FUNCTION_BLOCK SchieberVerriegelung (* Schieber verriegeln bei 3 Schieber *)
  (* Standard: 61499-2; Description: Copyright (c) 2025 HR Agrartechnik GmbH This program and the accompanying materials are made available under the terms of the Eclipse Public License 2.0 which is available at https://www.eclipse.org/legal/epl-2.0/ SPDX-License-Identifier: EPL-2.0 *)
  (* Version 1.0, 2025-06-04, Franz Höpfinger, HR Agrartechnik GmbH *)
  PACKAGE logiBUS::utils::sequence::schieber;
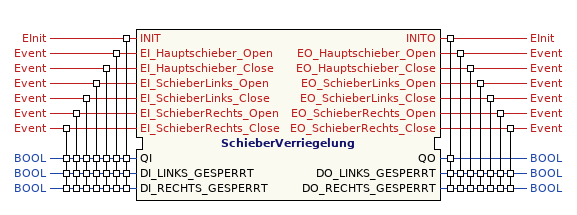
  EVENT_INPUT
    INIT : EInit WITH QI, DI_LINKS_GESPERRT, DI_RECHTS_GESPERRT; (* Initialization Request *)
    EI_Hauptschieber_Open WITH QI, DI_LINKS_GESPERRT, DI_RECHTS_GESPERRT;
    EI_Hauptschieber_Close WITH QI, DI_LINKS_GESPERRT, DI_RECHTS_GESPERRT;
    EI_SchieberLinks_Open WITH QI, DI_LINKS_GESPERRT, DI_RECHTS_GESPERRT;
    EI_SchieberLinks_Close WITH QI, DI_LINKS_GESPERRT, DI_RECHTS_GESPERRT;
    EI_SchieberRechts_Open WITH QI, DI_LINKS_GESPERRT, DI_RECHTS_GESPERRT;
    EI_SchieberRechts_Close WITH QI, DI_LINKS_GESPERRT, DI_RECHTS_GESPERRT;
  END_EVENT
  EVENT_OUTPUT
    INITO : EInit WITH QO, DO_LINKS_GESPERRT, DO_RECHTS_GESPERRT; (* Initialization Confirm *)
    EO_Hauptschieber_Open WITH DO_LINKS_GESPERRT, DO_RECHTS_GESPERRT;
    EO_Hauptschieber_Close WITH DO_LINKS_GESPERRT, DO_RECHTS_GESPERRT;
    EO_SchieberLinks_Open WITH DO_LINKS_GESPERRT, DO_RECHTS_GESPERRT;
    EO_SchieberLinks_Close WITH DO_LINKS_GESPERRT, DO_RECHTS_GESPERRT;
    EO_SchieberRechts_Open WITH DO_LINKS_GESPERRT, DO_RECHTS_GESPERRT;
    EO_SchieberRechts_Close WITH DO_LINKS_GESPERRT, DO_RECHTS_GESPERRT;
  END_EVENT
  VAR_INPUT
    QI : BOOL; (* Input event qualifier *)
    DI_LINKS_GESPERRT : BOOL;
    DI_RECHTS_GESPERRT : BOOL;
  END_VAR
  VAR_OUTPUT
    QO : BOOL; (* Output event qualifier *)
    DO_LINKS_GESPERRT : BOOL;
    DO_RECHTS_GESPERRT : BOOL;
  END_VAR
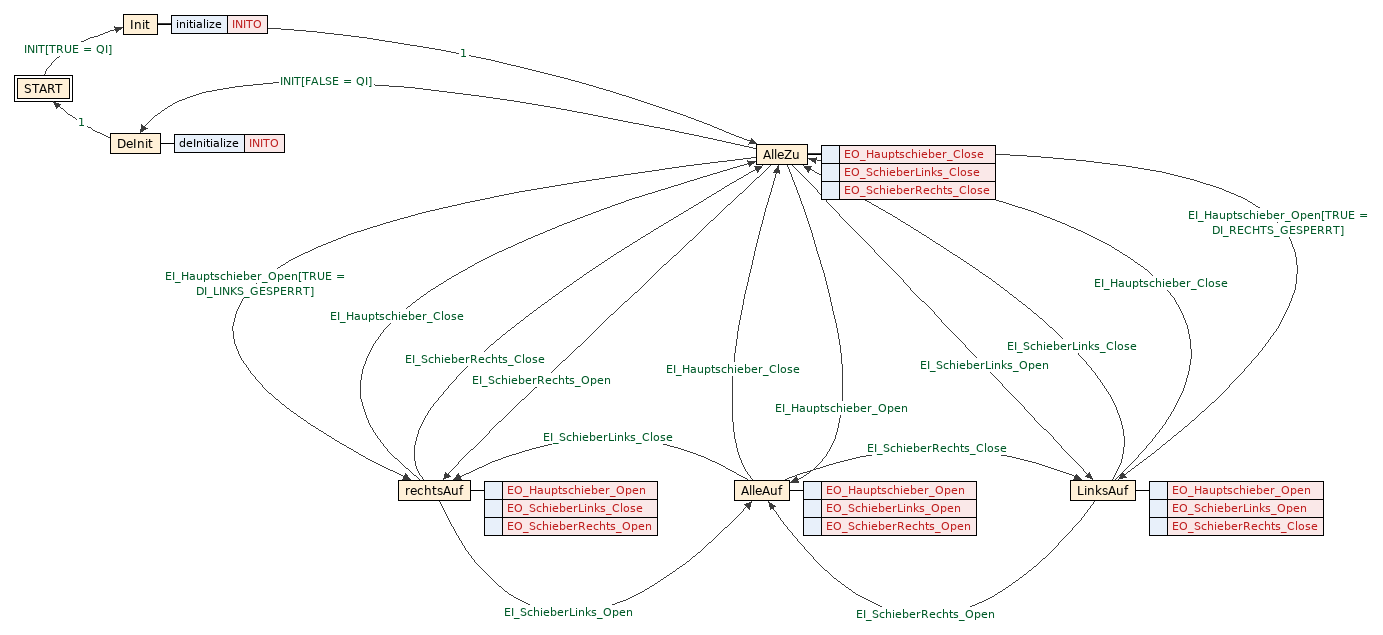
  EC_STATES
    START; (* Initial State *)
    Init : initialize -> INITO; (* Initialization *)
    DeInit : deInitialize -> INITO;
    AlleZu : -> EO_Hauptschieber_Close, -> EO_SchieberLinks_Close, -> EO_SchieberRechts_Close;
    AlleAuf : -> EO_Hauptschieber_Open, -> EO_SchieberLinks_Open, -> EO_SchieberRechts_Open;
    LinksAuf : -> EO_Hauptschieber_Open, -> EO_SchieberLinks_Open, -> EO_SchieberRechts_Close;
    rechtsAuf : -> EO_Hauptschieber_Open, -> EO_SchieberLinks_Close, -> EO_SchieberRechts_Open;
  END_STATES
  EC_TRANSITIONS
    START TO Init := INIT[TRUE = QI];
    DeInit TO START := 1;
    AlleZu TO rechtsAuf := EI_SchieberRechts_Open;
    AlleZu TO LinksAuf := EI_SchieberLinks_Open;
    rechtsAuf TO AlleZu := EI_SchieberRechts_Close;
    LinksAuf TO AlleZu := EI_SchieberLinks_Close;
    LinksAuf TO AlleAuf := EI_SchieberRechts_Open;
    rechtsAuf TO AlleAuf := EI_SchieberLinks_Open;
    AlleAuf TO rechtsAuf := EI_SchieberLinks_Close;
    AlleAuf TO LinksAuf := EI_SchieberRechts_Close;
    AlleAuf TO AlleZu := EI_Hauptschieber_Close;
    rechtsAuf TO AlleZu := EI_Hauptschieber_Close;
    LinksAuf TO AlleZu := EI_Hauptschieber_Close;
    AlleZu TO DeInit := INIT[FALSE = QI];
    Init TO AlleZu := 1;
    AlleZu TO LinksAuf := EI_Hauptschieber_Open[TRUE = DI_RECHTS_GESPERRT];
    AlleZu TO rechtsAuf := EI_Hauptschieber_Open[TRUE = DI_LINKS_GESPERRT];
    AlleZu TO AlleAuf := EI_Hauptschieber_Open;
  END_TRANSITIONS
  ALGORITHM initialize IN ST:
QO := QI;
  END_ALGORITHM
  ALGORITHM deInitialize IN ST:
QO := FALSE;
  END_ALGORITHM
  ALGORITHM normalOperation IN ST:
QO := QI;

IF TRUE = QI THEN
	(* only perform normal operation of QI is true *)
	DO_LINKS_GESPERRT := DI_LINKS_GESPERRT;
	DO_RECHTS_GESPERRT := DI_RECHTS_GESPERRT;

END_IF;
  END_ALGORITHM
END_FUNCTION_BLOCK
